PROGRAM MAIN
VAR
	stThisIsFirstEvent: ST_Event;
	bBoolean: BOOL :=FALSE;
	bBoolean_2: BOOL :=FALSE;
END_VAR

IF NOT bBoolean THEN
UpdateEventWithSystemTime(stEvent:= stThisIsFirstEvent);
bBoolean := TRUE;
END_IF

END_PROGRAM

(* stored: Version 1.1.0.1, ProductVersion 3.1.4024.12
   POU MAIN: Id {60c21c48-0c32-4eb0-bb4d-b2a6ceb38ded}, SpecialFunc None *)
